FUNCTION F_SCANNER_OpState : BYTE
VAR_INPUT
	bEnable				: BOOL;
	bConfigMode			: BOOL;
	bCodeChangeActive	: BOOL;
	bScannerReady		: BOOL;
END_VAR
VAR
END_VAR
(*
-------------------------------------------------------------------------------------------------
DATE		Version	Author	Comments
-------------------------------------------------------------------------------------------------
30/01/2015	3.00.00	PB		Initial release
							0 = Grey, disabled or offline
							1 = Blue, configuration mode active
							2 = Red, alarm active or comms loss
							3 = Orange, external condition off
							4 = Yellow, warning active
							5 = Green, operational

-------------------------------------------------------------------------------------------------
*)

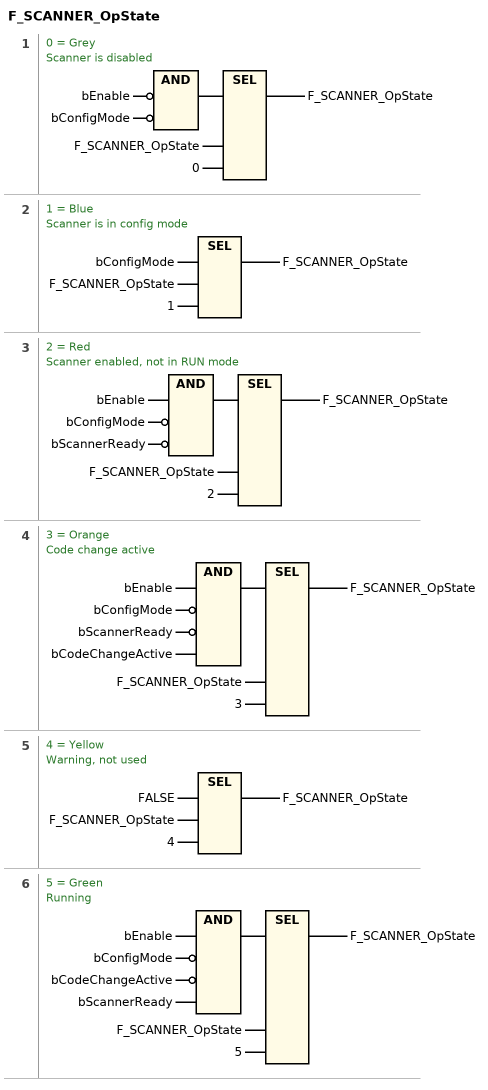
// NETWORK 1
// 					0 = Grey
// Scanner is disabled
//
F_SCANNER_OpState := SEL(NOT bEnable AND NOT bConfigMode, F_SCANNER_OpState, 0);

// NETWORK 2
// 					1 = Blue
// Scanner is in config mode
//
F_SCANNER_OpState := SEL(bConfigMode, F_SCANNER_OpState, 1);

// NETWORK 3
// 					2 = Red
// Scanner enabled, not in RUN mode
//
F_SCANNER_OpState := SEL(bEnable AND NOT bConfigMode AND NOT bScannerReady, F_SCANNER_OpState, 2);

// NETWORK 4
// 					3 = Orange
// Code change active
//
F_SCANNER_OpState := SEL(bEnable AND NOT bConfigMode AND NOT bScannerReady AND bCodeChangeActive, F_SCANNER_OpState, 3);

// NETWORK 5
// 					4 = Yellow
// Warning, not used
//
F_SCANNER_OpState := SEL(FALSE, F_SCANNER_OpState, 4);

// NETWORK 6
// 					5 = Green
// Running
//
F_SCANNER_OpState := SEL(bEnable AND NOT bConfigMode AND NOT bCodeChangeActive AND bScannerReady, F_SCANNER_OpState, 5);

END_FUNCTION

(* stored: Version 1.1.0.1, ProductVersion 3.1.4024.15
   POU F_SCANNER_OpState: Id {b08cca56-4834-493a-b78d-a85053314063}, SpecialFunc None *)
